Staubli VAL3: onF3Event.pgx

program onF3Event()
  local tool l_tTool
begin
  // look if the bButton is enable
  if bButton[2]
    //
    // get the tool
    call tcp:getTool(tTool,saveData:nFrameTool)
    if nFrame>0
      call use:timerDialog("Frame "+sEvent+" actived",3)
      fSetFrame.trsf=saveData:fFrameItem[nFrame].fFrame.trsf
    else
      call use:timerDialog("WORLD Frame actived",3)
      fSetFrame=world
    endIf
    $jogContext(tTool,fSetFrame,0)
    // save the  actual frame
    saveData:nFrameActive=nFrame
  endIf
end
